Yaskawa INFORM job: KRIS2(-160_-90)34.JBI

/JOB
//NAME KRIS2(-160_-90)34
//POS
///NPOS 148,148,148,10,0,0
///TOOL 0
///POSTYPE PULSE
///PULSE
C00000=-136908,-99459,-124829,20670,71348,76391
C00001=-134470,-76528,-106815,19279,71473,77234
C00002=-159578,-94739,-111578,14965,102577,71346
C00003=-157566,-87256,-71357,3912,80960,68626
C00004=-136911,-97837,-71335,2043,74746,75596
C00005=-137353,-98864,-69097,2107,72853,75411
C00006=-137353,-97788,-67030,2113,72134,75401
C00007=-137490,-98681,-67551,2126,71999,75348
C00008=-137823,-100474,-68178,2166,71474,75224
C00009=-137490,-99527,-69160,2120,72554,75357
C00010=-137490,-112967,-99500,2043,84312,75553
C00011=-132962,-68022,-80970,1616,95894,77239
C00012=-133097,-70190,-77189,1618,92458,77150
C00013=-133258,-72060,-76849,1633,91294,77082
C00014=-133258,-72050,-75890,1633,90711,77076
C00015=-133258,-72054,-76082,1633,90828,77076
C00016=-133486,-74582,-77287,1655,90276,76993
C00017=-133258,-72036,-78289,1635,92195,77094
C00018=-140979,-108094,-110643,2385,93763,74547
C00019=-136708,-68987,-94400,2043,103743,76128
C00020=-131299,-72562,-92979,1477,100921,77847
C00021=-133146,-74049,-93072,1658,100250,77236
C00022=-133146,-74446,-92238,1656,99534,77226
C00023=-133146,-74366,-92413,1656,99682,77228
C00024=-133350,-76932,-93602,1669,99101,77153
C00025=-133146,-73112,-94745,1670,101761,77256
C00026=-154612,-58853,-87611,3798,105373,70356
C00027=-154636,-59803,-86532,3777,104225,70312
C00028=-154636,-60502,-85461,3758,103210,70280
C00029=-154636,-60414,-85604,3761,103342,70284
C00030=-155113,-62506,-86695,3797,102960,70115
C00031=-154600,-59756,-86288,3773,104099,70317
C00032=-161369,-86849,-99090,4273,98390,67906
C00033=-162299,-90705,-86659,4280,88832,67270
C00034=-162680,-91589,-85702,4311,87811,67106
C00035=-162680,-91368,-84537,4311,87211,67083
C00036=-162680,-91407,-84732,4311,87310,67086
C00037=-163568,-93888,-85727,4385,86696,66764
C00038=-162680,-92039,-88633,4311,89381,67156
C00039=-171854,-115132,-97044,5055,83246,63813
C00040=-176135,-99923,-70409,842,76306,62354
C00041=-176746,-100127,-69456,876,75622,62141
C00042=-176746,-99180,-67670,877,75010,62140
C00043=-176746,-99324,-67941,877,75103,62140
C00044=-178145,-101177,-68585,955,74562,61655
C00045=-175862,-99037,-69317,825,76087,62452
C00046=-145436,-132582,-96247,-390,75065,72870
C00047=-166235,-131980,-119843,4599,88258,65923
C00048=-156260,-82084,-105550,20461,72444,69801
C00049=-137260,-84248,-120477,10166,77039,76482
C00050=-137260,-138866,-133764,10166,31487,76482
C00051=-31464,-162597,-133764,10166,12061,76482
C00052=11401,-148032,-125425,11667,35640,75771
C00053=126225,-114648,-117375,36487,17100,65054
C00054=160935,-140983,-109640,13468,75088,74332
C00055=169853,-118963,-84593,12681,69660,-86771
C00056=108998,-121589,-78490,-3111,72246,-67652
C00057=101498,-120645,-75827,-2941,70822,-70188
C00058=101498,-119392,-74038,-2947,70366,-70178
C00059=101498,-119562,-74281,-2946,70428,-70180
C00060=100817,-121900,-74755,-2942,69496,-70390
C00061=101437,-120901,-75918,-2941,70745,-70208
C00062=101671,-144527,-108100,-2850,78408,-70309
C00063=107420,-98138,-90760,-2968,91765,-68662
C00064=106123,-97431,-89210,-2933,91127,-69086
C00065=106079,-97593,-88323,-2932,90500,-69086
C00066=106079,-97314,-87194,-2931,89950,-69074
C00067=106079,-97371,-87421,-2931,90060,-69077
C00068=105757,-100151,-88472,-2922,89269,-69167
C00069=106110,-97559,-89281,-2933,91108,-69092
C00070=106110,-97729,-106489,-3015,101600,-69341
C00071=107817,-77200,-97797,-1990,101006,-68606
C00072=107961,-76698,-94617,-1993,99314,-68531
C00073=107961,-77099,-93736,-1989,98568,-68519
C00074=107961,-77014,-93933,-1989,98733,-68521
C00075=107703,-80198,-95370,-1956,97976,-68594
C00076=107832,-78083,-95841,-1978,99355,-68573
C00077=108708,-76271,-95015,4538,100749,-88680
C00078=108939,-78492,-94449,4493,99251,-88659
C00079=149006,-93113,-100988,-5479,101691,-74295
C00080=149599,-96300,-103483,-5484,101628,-74092
C00081=108723,-78074,-94057,-3078,98267,-89791
C00082=113965,-80387,-98246,-3646,99862,-88118
C00083=112015,-122483,-114020,-3369,87877,-88431
C00084=116962,-114728,-95357,-3904,80614,-86540
C00085=117676,-115580,-93267,-3992,78929,-86241
C00086=163022,-96736,-99152,22139,103253,-76925
C00087=162158,-93804,-96763,22109,103515,-77196
C00088=104974,-113131,-92422,-2667,79138,-90618
C00089=109141,-112938,-93941,-3100,80321,-89215
C00090=113958,-156480,-105404,-3885,65233,-87099
C00091=113958,-135498,-81926,-4007,61575,-86972
C00092=116417,-133537,-76878,-4367,59600,-86012
C00093=163006,-94576,-83573,21494,95359,-78388
C00094=162142,-91714,-81191,21448,95589,-78662
C00095=102513,-131504,-76174,-5344,59166,-90609
C00096=115088,-145817,-91151,-6745,61908,-86191
C00097=120295,-145940,-91152,-7309,62276,-84335
C00098=149731,-158641,-113843,14975,70738,69794
C00099=149731,-158641,-113843,14975,70738,69794
C00100=126225,-114648,-117375,36487,17100,65054
C00101=118781,-153853,-134406,32592,23357,65054
C00102=12470,-167083,-125425,11667,16324,75771
C00103=-137258,-84249,-120477,10166,64820,76482
C00104=-160540,-100857,-113063,23155,68829,67581
C00105=-144636,-173309,-129138,11293,64944,72208
C00106=-135566,-152591,-120530,7709,74393,76314
C00107=-139328,-137243,-114591,7038,82665,75517
C00108=-158743,-95268,-103371,5812,102972,69826
C00109=-157888,-92366,-100981,5813,102933,70115
C00110=-124816,-141390,-115691,5849,80052,80369
C00111=-126467,-143470,-120820,5933,82464,79916
C00112=-128645,-195873,-132590,6758,63059,78142
C00113=-144821,-162395,-106929,7940,65866,72581
C00114=-148359,-160820,-103988,8227,65211,71287
C00115=-158755,-94787,-86481,-976,103949,69303
C00116=-157900,-91912,-84097,-841,103969,69603
C00117=-127169,-165255,-104679,6709,61510,78579
C00118=-127169,-170980,-109668,6701,61638,78586
C00119=-127203,-187747,-112013,6590,55501,77611
C00120=-134083,-168892,-86258,-5,48650,76638
C00121=-143148,-164345,-80155,959,47272,73295
C00122=-158782,-86330,-62292,2348,97119,70521
C00123=-157926,-83586,-59872,2521,97014,70811
C00124=-112444,-165239,-80141,1803,46689,83534
C00125=-112444,-177354,-90291,1803,46710,83534
C00126=-133031,-170450,-89431,-9055,52143,79525
C00127=-144276,-143837,-77307,-9784,64447,75054
C00128=-158743,-95268,-103371,5812,102972,69826
C00129=-157888,-92366,-100981,5813,102933,70115
C00130=-165638,-137741,-76392,-10108,64585,67776
C00131=-153062,-184084,-115520,-9876,66274,71927
C00132=-133135,-130401,-99458,-8486,85928,77222
C00133=-133135,-130401,-99458,-8486,85928,77222
C00134=-135551,-131434,-96547,-8621,83375,76573
C00135=-158755,-94787,-86481,-976,103949,69303
C00136=-157900,-91912,-84097,-841,103969,69603
C00137=-150058,-125759,-94981,-9096,83717,71597
C00138=-150058,-139901,-119688,-9083,91560,71028
C00139=-133476,-138679,-117533,-8523,92690,76646
C00140=-134425,-135159,-113251,-8558,91771,76382
C00141=-158782,-86330,-62292,2348,97119,70521
C00142=-157926,-83586,-59872,2521,97014,70811
C00143=-147900,-127910,-111147,-9048,92698,71685
C00144=-139154,-141635,-132500,-8927,99684,74194
C00145=-159578,-94739,-111578,14965,102577,71346
C00146=-134470,-76528,-106815,19279,71473,77234
C00147=-36470,-76528,-106815,19279,71473,77234
BC00000=353535,857279,1075175
BC00001=353535,895977,1075175
BC00002=353535,975867,1075175
BC00003=382950,976989,1075175
BC00004=382950,976989,1075175
BC00005=382950,976989,1075175
BC00006=382950,976989,1075175
BC00007=382950,976989,1075172
BC00008=382950,976989,1075172
BC00009=382950,976989,1075172
BC00010=382950,976989,1075172
BC00011=382950,976989,1075172
BC00012=382950,976989,1075172
BC00013=382950,976989,1075172
BC00014=382950,976989,1075172
BC00015=382950,976989,1075172
BC00016=382950,976989,1075172
BC00017=382950,976989,1075172
BC00018=382092,1006363,1075175
BC00019=382092,1006363,1075175
BC00020=382092,1006363,1075175
BC00021=382092,1006363,1075175
BC00022=382092,1006363,1075175
BC00023=382092,1006363,1075175
BC00024=382092,1006363,1075175
BC00025=382092,1006363,1075175
BC00026=324712,1006363,1075175
BC00027=324712,1006363,1075175
BC00028=324712,1006363,1075175
BC00029=324712,1006363,1075175
BC00030=324712,1006363,1075175
BC00031=324712,1006363,1075175
BC00032=324712,1006363,1075175
BC00033=324712,1006363,1075175
BC00034=324712,1006363,1075175
BC00035=324712,1006363,1075175
BC00036=324712,1006363,1075175
BC00037=324712,1006363,1075175
BC00038=324712,1006363,1075175
BC00039=324712,1006363,1075175
BC00040=335336,1006363,1075175
BC00041=335336,1006363,1075175
BC00042=335336,1006363,1075175
BC00043=335336,1006363,1075175
BC00044=335336,1006363,1075175
BC00045=335336,1006363,1075175
BC00046=334035,1006363,1075175
BC00047=382070,1033391,1075175
BC00048=381896,966588,1075175
BC00049=353816,923989,1075175
BC00050=353816,923989,1075175
BC00051=379773,1126391,1075175
BC00052=398190,1030285,1075175
BC00053=312632,1138057,1075175
BC00054=340753,1115300,1075175
BC00055=340766,1114848,1075175
BC00056=340766,1114848,1075171
BC00057=340766,1114849,1075169
BC00058=340766,1114849,1075169
BC00059=340766,1114849,1075169
BC00060=340766,1114849,1075169
BC00061=340766,1114849,1075169
BC00062=340766,1114849,1075169
BC00063=340766,1114849,1075169
BC00064=340766,1114849,1075169
BC00065=340766,1114849,1075169
BC00066=340766,1114849,1075169
BC00067=340766,1114849,1075169
BC00068=340766,1114849,1075169
BC00069=340766,1114849,1075169
BC00070=340766,1114849,1075169
BC00071=340766,1114849,1075169
BC00072=340766,1114849,1075169
BC00073=340766,1114849,1075169
BC00074=340766,1114849,1075169
BC00075=340766,1114849,1075169
BC00076=340766,1114849,1075169
BC00077=340766,1114849,1075169
BC00078=340766,1114849,1075169
BC00079=348912,1090234,1075175
BC00080=348912,1090234,1075175
BC00081=340766,1114849,1075169
BC00082=340766,1114849,1075169
BC00083=340766,1114849,1075169
BC00084=340766,1114849,1075169
BC00085=340766,1114849,1075169
BC00086=322536,1051450,1075175
BC00087=322536,1051450,1075175
BC00088=340766,1114849,1075169
BC00089=340766,1114849,1075169
BC00090=340766,1114849,1075169
BC00091=340766,1114849,1075169
BC00092=340766,1114849,1075169
BC00093=322462,1078251,1075175
BC00094=322462,1078251,1075175
BC00095=340766,1114849,1075169
BC00096=340766,1114849,1075169
BC00097=340766,1114849,1075169
BC00098=340753,1115300,1075175
BC00099=340753,1115300,1075175
BC00100=312632,1138057,1075175
BC00101=312632,1138057,1075175
BC00102=398190,1030285,1075175
BC00103=353817,923990,1075175
BC00104=381896,966588,1075175
BC00105=363636,1044565,1075175
BC00106=363636,1044565,1075175
BC00107=363636,1044565,1075175
BC00108=364655,1041006,1075175
BC00109=364655,1041006,1075175
BC00110=363636,1044565,1075175
BC00111=363939,1044416,1075175
BC00112=363939,1044416,1075175
BC00113=363939,1044416,1075175
BC00114=363939,1044416,1075175
BC00115=364774,1039056,1075175
BC00116=364774,1039056,1075175
BC00117=363939,1044416,1075175
BC00118=363939,1044416,1075175
BC00119=363939,1044416,1075175
BC00120=363939,1044416,1075175
BC00121=363939,1044416,1075175
BC00122=355520,1012445,1075175
BC00123=355520,1012445,1075175
BC00124=363939,1044416,1075175
BC00125=363939,1044416,1075175
BC00126=304242,1044416,1075175
BC00127=304242,1044416,1075175
BC00128=364655,1041006,1075175
BC00129=364655,1041006,1075175
BC00130=304242,1044416,1075175
BC00131=304242,1044416,1075175
BC00132=304242,1044416,1075175
BC00133=304242,1044416,1075175
BC00134=304242,1044416,1075175
BC00135=364774,1039056,1075175
BC00136=364774,1039056,1075175
BC00137=304242,1044416,1075175
BC00138=304242,1044416,1075175
BC00139=304242,1065221,1075175
BC00140=304242,1065221,1075175
BC00141=355520,1012445,1075175
BC00142=355520,1012445,1075175
BC00143=304242,1065221,1075175
BC00144=304242,1065221,1075175
BC00145=353535,975867,1075175
BC00146=353535,895977,1075175
BC00147=295325,674563,1075175
EC00000=-1418945,-556475
EC00001=-1418945,-556475
EC00002=-1418945,-556475
EC00003=-1418945,-556475
EC00004=-1418945,-556475
EC00005=-1418945,-556475
EC00006=-1418945,-556475
EC00007=-1418944,-556475
EC00008=-1418944,-556475
EC00009=-1418944,-556475
EC00010=-1418944,-556475
EC00011=-1418944,-556475
EC00012=-1418944,-556475
EC00013=-1418944,-556475
EC00014=-1418944,-556475
EC00015=-1418944,-556475
EC00016=-1418944,-556475
EC00017=-1418944,-556475
EC00018=-1418945,-556475
EC00019=-1418945,-556475
EC00020=-1418945,-556475
EC00021=-1418945,-556475
EC00022=-1418945,-556475
EC00023=-1418945,-556475
EC00024=-1418945,-556475
EC00025=-1418945,-556475
EC00026=-1418945,-556475
EC00027=-1418945,-556475
EC00028=-1418945,-556475
EC00029=-1418945,-556475
EC00030=-1418945,-556475
EC00031=-1418945,-556475
EC00032=-1418945,-556475
EC00033=-1418945,-556475
EC00034=-1418945,-556475
EC00035=-1418945,-556475
EC00036=-1418945,-556475
EC00037=-1418945,-556475
EC00038=-1418945,-556475
EC00039=-1418945,-556475
EC00040=-1418945,-556475
EC00041=-1418945,-556475
EC00042=-1418945,-556475
EC00043=-1418945,-556475
EC00044=-1418945,-556475
EC00045=-1418945,-556475
EC00046=-1418945,-556475
EC00047=-1418945,-556475
EC00048=-1418945,-556475
EC00049=-1418945,-556475
EC00050=-1418945,-556475
EC00051=-1418945,-556475
EC00052=-1595090,-3837
EC00053=-1773681,556475
EC00054=-1773681,556475
EC00055=-1773681,556475
EC00056=-1773682,556473
EC00057=-1773683,556473
EC00058=-1773683,556473
EC00059=-1773683,556473
EC00060=-1773683,556473
EC00061=-1773683,556473
EC00062=-1773683,556473
EC00063=-1773683,556473
EC00064=-1773683,556473
EC00065=-1773683,556473
EC00066=-1773683,556473
EC00067=-1773683,556473
EC00068=-1773683,556473
EC00069=-1773683,556473
EC00070=-1773683,556473
EC00071=-1773683,556473
EC00072=-1773683,556473
EC00073=-1773683,556473
EC00074=-1773683,556473
EC00075=-1773683,556473
EC00076=-1773683,556473
EC00077=-1773683,556473
EC00078=-1773683,556473
EC00079=-1773681,556475
EC00080=-1773681,556475
EC00081=-1773683,556473
EC00082=-1773683,556473
EC00083=-1773683,556473
EC00084=-1773683,556473
EC00085=-1773683,556473
EC00086=-1773681,556475
EC00087=-1773681,556475
EC00088=-1773683,556473
EC00089=-1773683,556473
EC00090=-1773683,556473
EC00091=-1773683,556473
EC00092=-1773683,556473
EC00093=-1773681,556475
EC00094=-1773681,556475
EC00095=-1773683,556473
EC00096=-1773683,556473
EC00097=-1773683,556473
EC00098=-1773681,556475
EC00099=-1773681,556475
EC00100=-1773681,556475
EC00101=-1773681,556475
EC00102=-1595090,-3837
EC00103=-1418947,-556468
EC00104=-1418945,-556475
EC00105=-1418945,-556475
EC00106=-1418945,-556475
EC00107=-1418945,-556475
EC00108=-1418945,-556475
EC00109=-1418945,-556475
EC00110=-1418945,-556475
EC00111=-1418945,-556475
EC00112=-1418945,-556475
EC00113=-1418945,-556475
EC00114=-1418945,-556475
EC00115=-1418945,-556475
EC00116=-1418945,-556475
EC00117=-1418945,-556475
EC00118=-1418945,-556475
EC00119=-1418945,-556475
EC00120=-1418945,-556475
EC00121=-1418945,-556475
EC00122=-1418945,-556475
EC00123=-1418945,-556475
EC00124=-1418945,-556475
EC00125=-1418945,-556475
EC00126=-1418945,-556475
EC00127=-1418945,-556475
EC00128=-1418945,-556475
EC00129=-1418945,-556475
EC00130=-1418945,-556475
EC00131=-1418945,-556475
EC00132=-1418945,-556475
EC00133=-1418945,-556475
EC00134=-1418945,-556475
EC00135=-1418945,-556475
EC00136=-1418945,-556475
EC00137=-1418945,-556475
EC00138=-1418945,-556475
EC00139=-1418945,-556475
EC00140=-1418945,-556475
EC00141=-1418945,-556475
EC00142=-1418945,-556475
EC00143=-1418945,-556475
EC00144=-1418945,-556475
EC00145=-1418945,-556475
EC00146=-1418945,-556475
EC00147=-1418945,-556475
///POSTYPE BASE
///RECTAN
///RCONF 0,0,0,0,0,0,0,0,0,0,0,0,0,0,0,0,0,0,0,0,0,0,0,0
P00006=0.000,0.000,0.000,0.0000,0.0000,0.0000
P00021=-0.225,-6.128,-0.405,0.0000,0.0000,0.0000
P00022=0.232,-0.094,-1.480,0.0000,0.0000,0.0000
P00023=0.143,-0.036,0.682,0.0000,0.0000,0.0000
P00024=0.145,-0.552,1.326,0.0000,0.0000,0.0000
P00025=-2.003,0.006,0.728,0.0000,0.0000,0.0000
P00026=0.562,-0.002,-0.337,0.0000,0.0000,0.0000
P00031=1.853,-0.001,-1.549,0.0000,0.0000,0.0000
P00032=1.957,0.503,-7.217,0.0000,0.0000,0.0000
///RCONF 0,0,0,0,1,0,0,0,0,0,0,0,0,0,0,0,0,0,0,0,0,0,0,0
P00033=-0.123,0.612,-5.012,0.0000,0.0000,0.0000
//INST
///DATE 2024/12/10 19:39
///ATTR SC,RW
///GROUP1 RB1,BS1
///GROUP2 ST1
NOP
MOVJ C00000 BC00000 VJ=100.00  +MOVJ EC00000 VJ=100.00
MOVJ C00001 BC00001 VJ=100.00  +MOVJ EC00001 VJ=100.00
MOVJ C00002 BC00002 VJ=100.00  +MOVJ EC00002 VJ=100.00
'Path S1422
SFTOF3D
MOVJ C00003 BC00003 VJ=100.00  +MOVJ EC00003 VJ=100.00
MOVL C00004 BC00004 V=400.0  +MOVJ EC00004 VJ=100.00
SMOVL C00005 BC00005 V=100.0  +MOVJ EC00005
SREFP 3 C00006 BC00006  +REFP EC00006
CALL JOB:SEARCH-R1-S13D
SET P021 P006
SFTON3D P021
SMOVL C00007 BC00007 V=100.0  +MOVJ EC00007
SREFP 3 C00008 BC00008  +REFP EC00008
CALL JOB:SEARCH-R1-S13D
SET P021 P006
SFTON3D P021
SMOVL C00009 BC00009 V=100.0  +MOVJ EC00009
MOVL C00010 BC00010 V=400.0  +MOVJ EC00010 VJ=100.00
MOVL C00011 BC00011 V=1000.0  +MOVJ EC00011 VJ=100.00
MOVJ C00012 BC00012 VJ=100.00  +MOVJ EC00012 VJ=100.00
'Path S1423
SFTOF3D
SMOVL C00013 BC00013 V=100.0  +MOVJ EC00013
SREFP 3 C00014 BC00014  +REFP EC00014
CALL JOB:SEARCH-R1-S13D
SET P022 P006
SFTON3D P022
SMOVL C00015 BC00015 V=100.0  +MOVJ EC00015
SREFP 3 C00016 BC00016  +REFP EC00016
CALL JOB:SEARCH-R1-S13D
SET P022 P006
SFTON3D P022
SMOVL C00017 BC00017 V=100.0  +MOVJ EC00017
MOVL C00018 BC00018 V=400.0  +MOVJ EC00018 VJ=100.00
MOVL C00019 BC00019 V=1000.0  +MOVJ EC00019 VJ=100.00
MOVJ C00020 BC00020 VJ=100.00  +MOVJ EC00020 VJ=100.00
'Path S1424
SFTOF3D
SMOVL C00021 BC00021 V=100.0  +MOVJ EC00021
SREFP 3 C00022 BC00022  +REFP EC00022
CALL JOB:SEARCH-R1-S13D
SET P023 P006
SFTON3D P023
SMOVL C00023 BC00023 V=100.0  +MOVJ EC00023
SREFP 3 C00024 BC00024  +REFP EC00024
CALL JOB:SEARCH-R1-S13D
SET P023 P006
SFTON3D P023
SMOVL C00025 BC00025 V=100.0  +MOVJ EC00025
MOVL C00026 BC00026 V=400.0  +MOVJ EC00026 VJ=100.00
SMOVL C00027 BC00027 V=100.0  +MOVJ EC00027
SREFP 3 C00028 BC00028  +REFP EC00028
CALL JOB:SEARCH-R1-S13D
SET P024 P006
SFTON3D P024
SMOVL C00029 BC00029 V=100.0  +MOVJ EC00029
SREFP 3 C00030 BC00030  +REFP EC00030
CALL JOB:SEARCH-R1-S13D
SET P024 P006
SFTON3D P024
SMOVL C00031 BC00031 V=100.0  +MOVJ EC00031
MOVL C00032 BC00032 V=400.0  +MOVJ EC00032 VJ=100.00
MOVL C00033 BC00033 V=1000.0  +MOVJ EC00033 VJ=100.00
'Path S1423
SFTOF3D
SMOVL C00034 BC00034 V=100.0  +MOVJ EC00034
SREFP 3 C00035 BC00035  +REFP EC00035
CALL JOB:SEARCH-R1-S13D
SET P025 P006
SFTON3D P025
SMOVL C00036 BC00036 V=100.0  +MOVJ EC00036
SREFP 3 C00037 BC00037  +REFP EC00037
CALL JOB:SEARCH-R1-S13D
SET P025 P006
SFTON3D P025
SMOVL C00038 BC00038 V=100.0  +MOVJ EC00038
MOVL C00039 BC00039 V=400.0  +MOVJ EC00039 VJ=100.00
MOVL C00040 BC00040 V=1000.0  +MOVJ EC00040 VJ=100.00
'Path S1424
SFTOF3D
SMOVL C00041 BC00041 V=100.0  +MOVJ EC00041
SREFP 3 C00042 BC00042  +REFP EC00042
CALL JOB:SEARCH-R1-S13D
SET P026 P006
SFTON3D P026
SMOVL C00043 BC00043 V=100.0  +MOVJ EC00043
SREFP 3 C00044 BC00044  +REFP EC00044
CALL JOB:SEARCH-R1-S13D
SET P026 P006
SFTON3D P026
SMOVL C00045 BC00045 V=100.0  +MOVJ EC00045
MOVL C00046 BC00046 V=400.0  +MOVJ EC00046 VJ=100.00
MOVL C00047 BC00047 V=1000.0  +MOVJ EC00047 VJ=100.00
'obrot
MOVJ C00048 BC00048 VJ=100.00  +MOVJ EC00048 VJ=100.00
MOVJ C00049 BC00049 VJ=100.00  +MOVJ EC00049 VJ=100.00
MOVJ C00050 BC00050 VJ=100.00  +MOVJ EC00050 VJ=100.00
MOVJ C00051 BC00051 VJ=100.00  +MOVJ EC00051 VJ=100.00
MOVJ C00052 BC00052 VJ=100.00  +MOVJ EC00052 VJ=100.00
MOVJ C00053 BC00053 VJ=100.00  +MOVJ EC00053 VJ=100.00
MOVJ C00054 BC00054 VJ=100.00  +MOVJ EC00054 VJ=100.00
'Path S1077
SFTOF3D
MOVJ C00055 BC00055 VJ=100.00  +MOVJ EC00055 VJ=100.00
MOVL C00056 BC00056 V=400.0  +MOVJ EC00056 VJ=100.00
SMOVL C00057 BC00057 V=100.0  +MOVJ EC00057
SREFP 3 C00058 BC00058  +REFP EC00058
CALL JOB:SEARCH-R1-S13D
SET P031 P006
SFTON3D P031
SMOVL C00059 BC00059 V=100.0  +MOVJ EC00059
SREFP 3 C00060 BC00060  +REFP EC00060
CALL JOB:SEARCH-R1-S13D
SET P031 P006
SFTON3D P031
SMOVL C00061 BC00061 V=100.0  +MOVJ EC00061
MOVL C00062 BC00062 V=1000.0  +MOVJ EC00062 VJ=100.00
MOVJ C00063 BC00063 VJ=100.00  +MOVJ EC00063 VJ=100.00
'Path S1078
SFTOF3D
MOVL C00064 BC00064 V=400.0  +MOVJ EC00064 VJ=100.00
SMOVL C00065 BC00065 V=100.0  +MOVJ EC00065
SREFP 3 C00066 BC00066  +REFP EC00066
CALL JOB:SEARCH-R1-S13D
SET P032 P006
SFTON3D P032
SMOVL C00067 BC00067 V=100.0  +MOVJ EC00067
SREFP 3 C00068 BC00068  +REFP EC00068
CALL JOB:SEARCH-R1-S13D
SET P032 P006
SFTON3D P032
SMOVL C00069 BC00069 V=100.0  +MOVJ EC00069
MOVL C00070 BC00070 V=1000.0  +MOVJ EC00070 VJ=100.00
'Path S1079
SFTOF3D
MOVL C00071 BC00071 V=400.0  +MOVJ EC00071 VJ=100.00
SMOVL C00072 BC00072 V=100.0  +MOVJ EC00072
SREFP 3 C00073 BC00073  +REFP EC00073
CALL JOB:SEARCH-R1-S13D
SET P033 P006
SFTON3D P033
SMOVL C00074 BC00074 V=100.0  +MOVJ EC00074
SREFP 3 C00075 BC00075  +REFP EC00075
CALL JOB:SEARCH-R1-S13D
SET P033 P006
SFTON3D P033
SMOVL C00076 BC00076 V=100.0  +MOVJ EC00076
SMOVL C00077 BC00077 V=166.7  +MOVJ EC00077
SFTON3D P033
SMOVL C00078 BC00078 V=133.3 PL=0  +MOVJ EC00078
SREFP 1 C00079 BC00079  +REFP EC00079
SREFP 2 C00080 BC00080  +REFP EC00080
MACRO1 MJ#(0) ARGF14
ARCON
SMOVL C00081 BC00081 V=10.0  +MOVJ EC00081
ARCOF
SMOVL C00082 BC00082 V=400.0  +MOVJ EC00082
SMOVL C00083 BC00083 V=1000.0  +MOVJ EC00083
SFTOF3D
MOVJ C00084 BC00084 VJ=100.00  +MOVJ EC00084 VJ=100.00
'Path W261
SFTOF3D
SFTON3D P032
SMOVL C00085 BC00085 V=133.3 PL=0  +MOVJ EC00085
SREFP 1 C00086 BC00086  +REFP EC00086
SREFP 2 C00087 BC00087  +REFP EC00087
MACRO1 MJ#(0) ARGF14
ARCON
SMOVL C00088 BC00088 V=10.0  +MOVJ EC00088
ARCOF
SMOVL C00089 BC00089 V=400.0  +MOVJ EC00089
SMOVL C00090 BC00090 V=1000.0  +MOVJ EC00090
SFTOF3D
'Path W1083
SFTOF3D
SFTON3D P031
MOVJ C00091 BC00091 VJ=100.00  +MOVJ EC00091 VJ=100.00
SMOVL C00092 BC00092 V=133.3 PL=0  +MOVJ EC00092
SREFP 1 C00093 BC00093  +REFP EC00093
SREFP 2 C00094 BC00094  +REFP EC00094
MACRO1 MJ#(0) ARGF14
ARCON
SMOVL C00095 BC00095 V=10.0  +MOVJ EC00095
ARCOF
SMOVL C00096 BC00096 V=400.0  +MOVJ EC00096
MOVJ C00097 BC00097 VJ=100.00  +MOVJ EC00097 VJ=50.00
'obrot
MOVJ C00098 BC00098 VJ=100.00  +MOVJ EC00098 VJ=100.00
MOVJ C00099 BC00099 VJ=100.00  +MOVJ EC00099 VJ=100.00
MOVJ C00100 BC00100 VJ=100.00  +MOVJ EC00100 VJ=100.00
MOVJ C00101 BC00101 VJ=100.00  +MOVJ EC00101 VJ=100.00
MOVJ C00102 BC00102 VJ=100.00  +MOVJ EC00102 VJ=100.00
MOVJ C00103 BC00103 VJ=100.00  +MOVJ EC00103 VJ=100.00
MOVJ C00104 BC00104 VJ=100.00  +MOVJ EC00104 VJ=100.00
'Path W1425
SFTOF3D
MOVJ C00105 BC00105 VJ=100.00  +MOVJ EC00105 VJ=100.00
SMOVL C00106 BC00106 V=166.7  +MOVJ EC00106
SFTON3D P023
SMOVL C00107 BC00107 V=133.3 PL=0  +MOVJ EC00107
SREFP 1 C00108 BC00108  +REFP EC00108
SREFP 2 C00109 BC00109  +REFP EC00109
MACRO1 MJ#(0) ARGF14
ARCON
SMOVL C00110 BC00110 V=10.0  +MOVJ EC00110
ARCOF
SMOVL C00111 BC00111 V=400.0  +MOVJ EC00111
SMOVL C00112 BC00112 V=1000.0  +MOVJ EC00112
SFTOF3D
'Path W1426
SFTOF3D
SFTON3D P022
MOVJ C00113 BC00113 VJ=100.00  +MOVJ EC00113 VJ=100.00
SMOVL C00114 BC00114 V=133.3 PL=0  +MOVJ EC00114
SREFP 1 C00115 BC00115  +REFP EC00115
SREFP 2 C00116 BC00116  +REFP EC00116
MACRO1 MJ#(0) ARGF14
ARCON
SMOVL C00117 BC00117 V=10.0  +MOVJ EC00117
ARCOF
SMOVL C00118 BC00118 V=400.0  +MOVJ EC00118
SMOVL C00119 BC00119 V=1000.0  +MOVJ EC00119
SFTOF3D
'Path W1427
SFTOF3D
SFTON3D P021
MOVJ C00120 BC00120 VJ=100.00  +MOVJ EC00120 VJ=100.00
SMOVL C00121 BC00121 V=133.3 PL=0  +MOVJ EC00121
SREFP 1 C00122 BC00122  +REFP EC00122
SREFP 2 C00123 BC00123  +REFP EC00123
MACRO1 MJ#(0) ARGF14
ARCON
SMOVL C00124 BC00124 V=10.0  +MOVJ EC00124
ARCOF
SMOVL C00125 BC00125 V=400.0  +MOVJ EC00125
SMOVL C00126 BC00126 V=166.7  +MOVJ EC00126
SFTON3D P026
SMOVL C00127 BC00127 V=133.3 PL=0  +MOVJ EC00127
SREFP 1 C00128 BC00128  +REFP EC00128
SREFP 2 C00129 BC00129  +REFP EC00129
MACRO1 MJ#(0) ARGF14
ARCON
SMOVL C00130 BC00130 V=10.0  +MOVJ EC00130
ARCOF
SMOVL C00131 BC00131 V=400.0  +MOVJ EC00131
SMOVL C00132 BC00132 V=1000.0  +MOVJ EC00132
SFTOF3D
'Path W1426
SFTOF3D
SFTON3D P025
MOVJ C00133 BC00133 VJ=100.00  +MOVJ EC00133 VJ=100.00
SMOVL C00134 BC00134 V=133.3 PL=0  +MOVJ EC00134
SREFP 1 C00135 BC00135  +REFP EC00135
SREFP 2 C00136 BC00136  +REFP EC00136
MACRO1 MJ#(0) ARGF14
ARCON
SMOVL C00137 BC00137 V=10.0  +MOVJ EC00137
ARCOF
SMOVL C00138 BC00138 V=400.0  +MOVJ EC00138
SMOVL C00139 BC00139 V=1000.0  +MOVJ EC00139
SFTOF3D
'Path W1427
SFTOF3D
SFTON3D P024
SMOVL C00140 BC00140 V=133.3 PL=0  +MOVJ EC00140
SREFP 1 C00141 BC00141  +REFP EC00141
SREFP 2 C00142 BC00142  +REFP EC00142
MACRO1 MJ#(0) ARGF14
ARCON
SMOVL C00143 BC00143 V=10.0  +MOVJ EC00143
ARCOF
SMOVL C00144 BC00144 V=400.0  +MOVJ EC00144
SFTOF3D
MOVJ C00145 BC00145 VJ=100.00  +MOVJ EC00145 VJ=100.00
MOVJ C00146 BC00146 VJ=100.00  +MOVJ EC00146 VJ=100.00
MOVJ C00147 BC00147 VJ=100.00  +MOVJ EC00147 VJ=100.00
END
